// TIA Portal V17 export
// export: Created 2025-08-05T09:36:00.5940405Z, ExportSetting WithDefaults, DisplayName Totally Integrated Automation Portal, DisplayVersion V17, DisplayName TIA Portal Openness, DisplayVersion V17, DisplayName TIA Portal Version Control Interface, DisplayVersion V17, DisplayName SINAMICS Startdrive Advanced, DisplayVersion V17, DisplayName SINAMICS Startdrive G130, G150, S120, S150, SINAMICS MV, S210, DisplayVersion V17, DisplayName SINAMICS Startdrive G110M, G120, G120C, G120D, G120P, G115D, DisplayVersion V17, DisplayName STEP 7 Professional, DisplayVersion V17, DisplayName STEP 7 Safety, DisplayVersion V17, DisplayName WinCC Advanced, DisplayVersion V17
TYPE "typeHmiOperatorPrompt"
// stored: IsFailsafeCompliant false
   STRUCT
      promt : Struct
         prompt1 : Bool;   // Bitte warten
         prompt2 : Bool;   // -
         prompt3 : Bool;   // -
         prompt4 : Bool;   // -
         prompt5 : Bool;   // Schweißmaskenwechsel - Montagehilfe nicht vorhanden
         prompt6 : Bool;   // Schweißmaskenwechsel - Schutztüre nicht geöffnet
         prompt7 : Bool;   // Schweißmaskenwechsel - DMC-Code Schweißmaske nicht korrekt
         prompt8 : Bool;   // Leistung ausschalten --> 'Start Aus'
         prompt9 : Bool;   // -
         prompt10 : Bool;   // Not-Halt Hauptbedienpult aufheben
         prompt11 : Bool;   // Not-Halt Mobile Panel aufheben
         prompt12 : Bool;   // Not-Halt Schutztüre 1 aufheben
         prompt13 : Bool;   // Not-Halt Schutztüre 2 aufheben
         prompt14 : Bool;   // Not-Halt Lasergerät 1 aufheben
         prompt15 : Bool;   // Not-Halt Lasergerät 2 aufheben
         prompt16 : Bool;   // Not-Halt Lasergerät 1 Bedienpult aufheben
         prompt17 : Bool;   // Not-Halt Lasergerät 1 Bedienpult aufheben
         prompt18 : Bool;   // -
         prompt19 : Bool;   // -
         prompt20 : Bool;   // Medien gesamt einschalten
         prompt21 : Bool;   // -
         prompt22 : Bool;   // -
         prompt23 : Bool;   // -
         prompt24 : Bool;   // Schutzeinrichtungen schliessen und verriegeln
         prompt25 : Bool;   // Schutztüre 1 schliessen
         prompt26 : Bool;   // Schutztüre 2 schliessen
         prompt27 : Bool;   // -
         prompt28 : Bool;   // -
         prompt29 : Bool;   // -
         prompt30 : Bool;   // Zustimmbetrieb nicht möglich --> mehr als eine Schutztür offen
         prompt31 : Bool;   // Zustimmtaste drücken
         prompt32 : Bool;   // -
         prompt33 : Bool;   // Leistungsmessgerät in Vorrichtung schieben und sichern
         prompt34 : Bool;   // Leistungsmessgerät und Beam-Watch in Vorrichtung schieben und sichern
         prompt35 : Bool;   // Opferblech Laser 1 ist verschlissen --> Wechseln
         prompt36 : Bool;   // Opferblech Laser 2 ist verschlissen --> Wechseln
         prompt37 : Bool;   // -
         prompt38 : Bool;   // -
         prompt39 : Bool;   // Leistung einschalten --> 'Start Ein'
         prompt40 : Bool;   // Start nicht möglich --> 'zur Grundstellung'
         prompt41 : Bool;   // Station starten --> 'Start'
         prompt42 : Bool;   // -
         prompt43 : Bool;   // -
         prompt44 : Bool;   // maximal eine Schutzeinrichtung öffnen/unterbrechen
         prompt45 : Bool;   // -
         prompt46 : Bool;   // -
         prompt47 : Bool;   // -
         prompt48 : Bool;   // -
         prompt49 : Bool;   // Start nicht möglich --> 'zur Grundstellung'
         prompt50 : Bool;   // Station starten --> 'Start'
         prompt51 : Bool;   // -
         prompt52 : Bool;   // -
         prompt53 : Bool;   // -
         prompt54 : Bool;   // -
         prompt55 : Bool;   // -
         prompt56 : Bool;   // -
         prompt57 : Bool;   // -
         prompt58 : Bool;   // -
         prompt59 : Bool;   // -
         prompt60 : Bool;   // -
         prompt61 : Bool;   // -
         prompt62 : Bool;   // -
         prompt63 : Bool;   // -
         prompt64 : Bool;   // Typwechsel quittieren
         prompt65 : Bool;   // SPR-Check ausführen und quittieren
         prompt66 : Bool;   // Missbrauchstest Stopp 1 erforderlich
         prompt67 : Bool;   // Missbrauchstest Stopp 2 erforderlich
         prompt68 : Bool;   // Missbrauchstest Stopp 3 erforderlich
         prompt69 : Bool;   // Missbrauchstest Stopp 4 erforderlich
         prompt70 : Bool;   // Missbrauchstest inaktiv (Zeit- und Stückzahlsteuerung deaktiviert)
         prompt71 : Bool;   // -
         prompt72 : Bool;   // -
         prompt73 : Bool;   // -
         prompt74 : Bool;   // Daten: Sicherungspuffer ist initial -> Daten sichern oder rücksichern!
         prompt75 : Bool;   // Daten Sicherung nicht aktuell
         prompt76 : Bool;   // Verschleißzähler: Sicherung ist initial -> Daten sichern oder rücksichern
         prompt77 : Bool;   // Verschleißzählerdaten nicht aktuell
         prompt78 : Bool;   // -
         prompt79 : Bool;   // -
         prompt80 : Bool;   // -
         prompt81 : Bool;   // -
         prompt82 : Bool;   // -
         prompt83 : Bool;   // -
         prompt84 : Bool;   // -
         prompt85 : Bool;   // -
         prompt86 : Bool;   // -
         prompt87 : Bool;   // -
         prompt88 : Bool;   // -
         prompt89 : Bool;   // -
         prompt90 : Bool;   // -
         prompt91 : Bool;   // -
         prompt92 : Bool;   // -
         prompt93 : Bool;   // -
         prompt94 : Bool;   // -
         prompt95 : Bool;   // -
         prompt96 : Bool;   // -
         prompt97 : Bool;   // -
         prompt98 : Bool;   // -
         prompt99 : Bool;   // -
         prompt100 : Bool;   // -
         prompt101 : Bool;   // -
         prompt102 : Bool;   // -
         prompt103 : Bool;   // -
         prompt104 : Bool;   // -
         prompt105 : Bool;   // -
         prompt106 : Bool;   // -
         prompt107 : Bool;   // -
         prompt108 : Bool;   // -
         prompt109 : Bool;   // -
         prompt110 : Bool;   // -
         prompt111 : Bool;   // -
         prompt112 : Bool;   // -
         prompt113 : Bool;   // -
         prompt114 : Bool;   // -
         prompt115 : Bool;   // -
         prompt116 : Bool;   // -
         prompt117 : Bool;   // -
         prompt118 : Bool;   // -
         prompt119 : Bool;   // -
         prompt120 : Bool;   // -
         prompt121 : Bool;   // -
         prompt122 : Bool;   // -
         prompt123 : Bool;   // -
         prompt124 : Bool;   // -
         prompt125 : Bool;   // -
         prompt126 : Bool;   // -
         prompt127 : Bool;   // -
         prompt128 : Bool;   // -
         prompt129 : Bool;   // -
         prompt130 : Bool;   // -
         prompt131 : Bool;   // -
         prompt132 : Bool;   // -
         prompt133 : Bool;   // -
         prompt134 : Bool;   // -
         prompt135 : Bool;   // -
         prompt136 : Bool;   // -
         prompt137 : Bool;   // -
         prompt138 : Bool;   // -
         prompt139 : Bool;   // -
         prompt140 : Bool;   // -
         prompt141 : Bool;   // -
         prompt142 : Bool;   // -
         prompt143 : Bool;   // -
         prompt144 : Bool;   // -
         prompt145 : Bool;   // -
         prompt146 : Bool;   // -
         prompt147 : Bool;   // -
         prompt148 : Bool;   // -
         prompt149 : Bool;   // -
         prompt150 : Bool;   // -
         prompt151 : Bool;   // -
         prompt152 : Bool;   // -
         prompt153 : Bool;   // -
         prompt154 : Bool;   // -
         prompt155 : Bool;   // -
         prompt156 : Bool;   // -
         prompt157 : Bool;   // -
         prompt158 : Bool;   // -
         prompt159 : Bool;   // -
         prompt160 : Bool;   // -
      END_STRUCT;
   END_STRUCT;
END_TYPE
